% RSLogix 500 project ELEVATOR 01( IN PROCESS)_BAK005.RSS, saved by version 8.30.00.16 %
PROJECT "UNTITLED"    % processor: Bul.1763 MicroLogix 1100 Series B %

PROGRAM FILES
  LAD 2   12 rungs

DATA FILES
  O0 OUTPUT  4 elements
  I1 INPUT  6 elements
  S2 STATUS  66 elements
  B3 BINARY  1 elements
  T4 TIMER  1 elements
  C5 COUNTER  1 elements
  R6 CONTROL  1 elements
  N7 INTEGER  1 elements
  F8 FLOAT  1 elements

LADDER 2
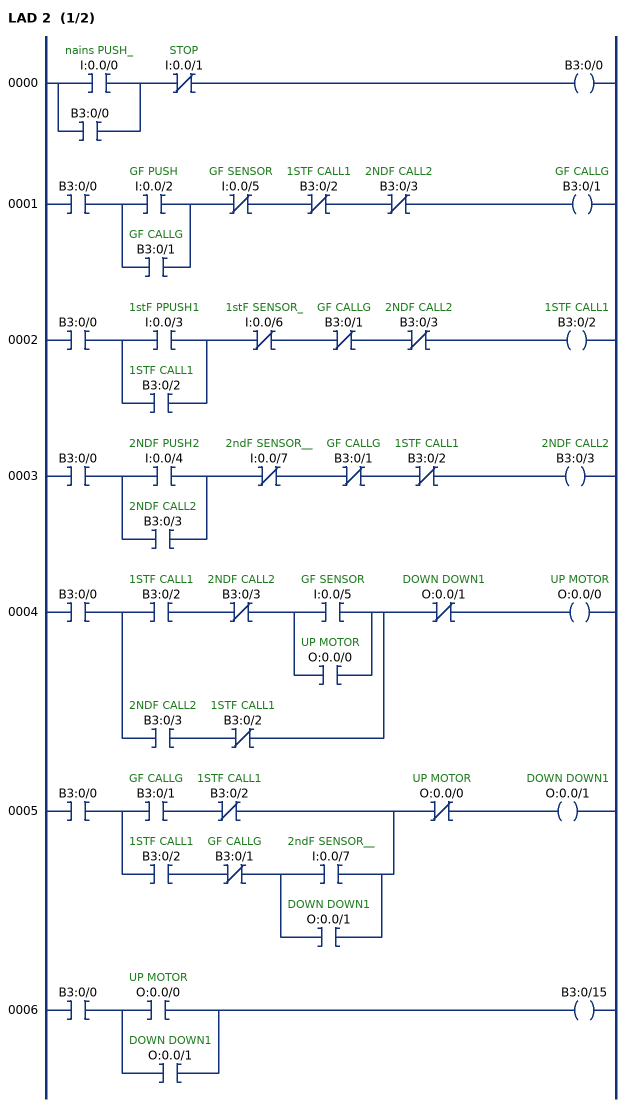
% Rung: 0 %
SOR BST XIC I:0.0/0 NXB XIC B3:0/0 BND XIO I:0.0/1 OTE B3:0/0 EOR
%   I:0.0/0  PUSH_  "nains" %
%   I:0.0/1  STOP %
% Rung: 1 %
SOR XIC B3:0/0 BST XIC I:0.0/2 NXB XIC B3:0/1 BND XIO I:0.0/5 XIO B3:0/2 XIO B3:0/3 OTE B3:0/1 EOR
%   I:0.0/2  PUSH  "GF" %
%   B3:0/1  CALLG  "GF" %
%   I:0.0/5  SENSOR  "GF" %
%   B3:0/2  CALL1  "1STF" %
%   B3:0/3  CALL2  "2NDF" %
% Rung: 2 %
SOR XIC B3:0/0 BST XIC I:0.0/3 NXB XIC B3:0/2 BND XIO I:0.0/6 XIO B3:0/1 XIO B3:0/3 OTE B3:0/2 EOR
%   I:0.0/3  PPUSH1  "1stF" %
%   B3:0/2  CALL1  "1STF" %
%   I:0.0/6  SENSOR_  "1stF" %
%   B3:0/1  CALLG  "GF" %
%   B3:0/3  CALL2  "2NDF" %
% Rung: 3 %
SOR XIC B3:0/0 BST XIC I:0.0/4 NXB XIC B3:0/3 BND XIO I:0.0/7 XIO B3:0/1 XIO B3:0/2 OTE B3:0/3 EOR
%   I:0.0/4  PUSH2  "2NDF" %
%   B3:0/3  CALL2  "2NDF" %
%   I:0.0/7  SENSOR__  "2ndF" %
%   B3:0/1  CALLG  "GF" %
%   B3:0/2  CALL1  "1STF" %
% Rung: 4 %
SOR XIC B3:0/0 BST XIC B3:0/2 XIO B3:0/3 BST XIC I:0.0/5 NXB XIC O:0.0/0 BND NXB XIC B3:0/3 XIO B3:0/2 BND XIO O:0.0/1 OTE O:0.0/0 EOR
%   B3:0/2  CALL1  "1STF" %
%   B3:0/3  CALL2  "2NDF" %
%   I:0.0/5  SENSOR  "GF" %
%   O:0.0/0  MOTOR  "UP" %
%   O:0.0/1  DOWN1  "DOWN" %
% Rung: 5 %
SOR XIC B3:0/0 BST XIC B3:0/1 XIO B3:0/2 NXB XIC B3:0/2 XIO B3:0/1 BST XIC I:0.0/7 NXB XIC O:0.0/1 BND BND XIO O:0.0/0 OTE O:0.0/1 EOR
%   B3:0/1  CALLG  "GF" %
%   B3:0/2  CALL1  "1STF" %
%   I:0.0/7  SENSOR__  "2ndF" %
%   O:0.0/1  DOWN1  "DOWN" %
%   O:0.0/0  MOTOR  "UP" %
% Rung: 6 %  % edit flag set %
SOR XIC B3:0/0 BST XIC O:0.0/0 NXB XIC O:0.0/1 BND OTE B3:0/15 EOR
%   O:0.0/0  MOTOR  "UP" %
%   O:0.0/1  DOWN1  "DOWN" %

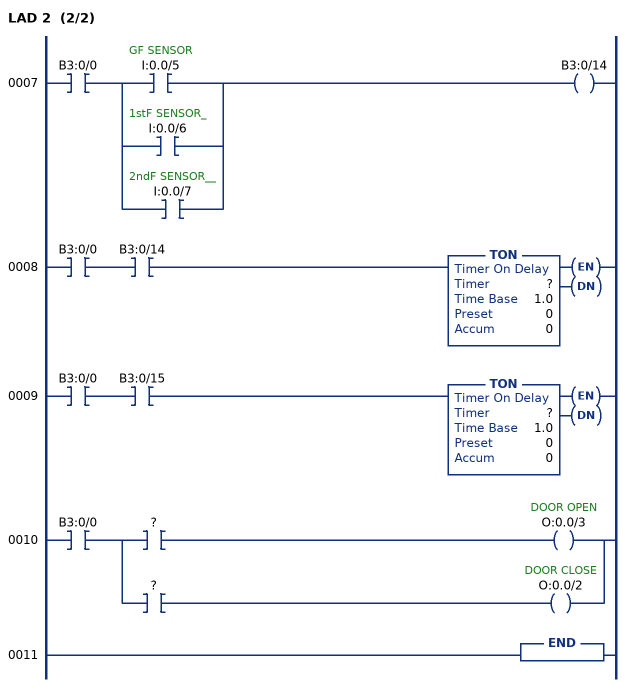
% Rung: 7 %  % edit flag set %
SOR XIC B3:0/0 BST XIC I:0.0/5 NXB XIC I:0.0/6 NXB XIC I:0.0/7 BND OTE B3:0/14 EOR
%   I:0.0/5  SENSOR  "GF" %
%   I:0.0/6  SENSOR_  "1stF" %
%   I:0.0/7  SENSOR__  "2ndF" %
% Rung: 8 %  % edit flag set %
SOR XIC B3:0/0 XIC B3:0/14 TON ? 1.0 0 0 EOR
% Rung: 9 %  % edit flag set %
SOR XIC B3:0/0 XIC B3:0/15 TON ? 1.0 0 0 EOR
% Rung: 10 %  % edit flag set %
SOR XIC B3:0/0 BST XIC ? OTE O:0.0/3 NXB XIC ? OTE O:0.0/2 BND EOR
%   O:0.0/3  OPEN  "DOOR" %
%   O:0.0/2  CLOSE  "DOOR" %
% Rung: 11 %
SOR END EOR

DATA TABLE (non-zero values as saved)
DATA B3
% B3:0 % 0X0001
